TYPE ST_RegDeadbandControls :
STRUCT
	(* Deadband controls *)
iDeadband	:	INT;
iMaxSpeed	:	INT; // degrees per second
END_STRUCT
END_TYPE

(* stored: Version 1.1.0.1, ProductVersion 3.1.0.24
   DUT ST_RegDeadbandControls: Id {a04513ee-c76f-4682-bef9-04f3920c05e2} *)
